// TIA Portal V17 export
// export: Created 2025-03-13T10:31:34.2201128Z, ExportSetting WithDefaults, DisplayName Totally Integrated Automation Portal, DisplayVersion V17 Update 8, DisplayName TIA Portal Openness, DisplayVersion V17 Update 8, DisplayName TIA Portal Version Control Interface, DisplayVersion V17, DisplayName SINAMICS Startdrive Advanced, DisplayVersion V17 SP2, DisplayName SINAMICS Startdrive G110M, G120, G120C, G120D, G120P, G115D, DisplayVersion V17 SP2, DisplayName SINAMICS Startdrive G130, G150, S120, S150, SINAMICS MV, S210, DisplayVersion V17 SP2, DisplayName STEP 7 Professional, DisplayVersion V17 Update 8, DisplayName SINUMERIK ONE STEP 7 Toolbox, DisplayVersion V17 Update 12, DisplayName SINUMERIK 840D sl STEP 7 Toolbox, DisplayVersion V17 Update 12, DisplayName STEP 7 Safety, DisplayVersion V17 Update 6, DisplayName WinCC Advanced, DisplayVersion V17 Update 8
TYPE "POWDER FEEDER HOPPER"
// stored: IsFailsafeCompliant false
   STRUCT
      "START GENERAL CONDITIONS" : Bool;
      "START INITIAL CONDITIONS" : Bool;
      "START MANUAL REQUEST" : Bool;
      "START AUTO REQUEST" : Bool;
      "START GLOBAL REQUESTE" : Bool;
      "START COMMAND" : Bool;
      START : Bool;
      "FEEDBACK ON" : Bool;
      "STOP GENERAL CONDITIONS" : Bool;
      "STOP INITIAL CONDITIONS" : Bool;
      "STOP MANUAL REQUEST" : Bool;
      "STOP AUTO REQUEST" : Bool;
      "STOP GLOBAL REQUEST" : Bool;
      "STOP COMMAND" : Bool;
      STOP : Bool;
      "FEEDBACK OFF" : Bool;
      "START GENERAL CONDITIONS HELP" : Bool;
      "START INITIAL CONDITIONS HELP" : Bool;
      "STOP GENERAL CONDITIONS HELP" : Bool;
      "STOP INITIAL CONDITIONS HELP" : Bool;
      FAULT : Bool;
   END_STRUCT;
END_TYPE
